// TIA Portal V19 export
TYPE "typeCanProcessImageOutputs"
   STRUCT
      SlaveDigitalOutput1 : Byte;
      SlaveDigitalOutput2 : Byte;
      SlaveAnalogOutput1 : Int;
      SlaveAnalogOutput2 : Int;
      SlaveAnalogOutput3 : Int;
      SlaveAnalogOutput4 : Int;
   END_STRUCT;
END_TYPE
